(* CoDeSys 2.3 export: F_READ_SENSOR_BAR.EXP *)

(* POU FUN/PARAMETERS/F_READ_SENSOR_BAR, ST *)
FUNCTION F_READ_SENSOR_BAR : BOOL
VAR_INPUT
END_VAR
VAR_IN_OUT
	stSensor : ST_SENSOR_BAR;
	fbIdList : FB_IDLIST;
END_VAR
VAR
END_VAR
stSensor.Cal_K   := F_IDLIST_GETREAL( CONCAT(stSensor.Name, '_K'   ), fbIdList );
stSensor.Cal_Off := stSensor.Cal_K * -stSensor.Raw_Off;
stSensor.MaxBar  := F_IDLIST_GETREAL( CONCAT(stSensor.Name, '_Max' ), fbIdList );
END_FUNCTION
